TYPE ST_KPI_CasePackerSignals :
STRUCT
	nSensor			: UDINT;
	nMachine		: UDINT;
	nPLC			: UDINT;

END_STRUCT
END_TYPE

(* stored: Version 1.1.0.1
   DUT ST_KPI_CasePackerSignals: Id {cfc09ba3-0c4e-4372-99c3-ed9d43b1738d} *)
